Staubli VAL3: isReachable.pgx

program isReachable(pointRx& x_pPoint[], tool x_tTool, bool& x_bUnreached)
  local joint l_jJoint
  local point l_pPoint
begin
  // check the point...
  if pointToJoint(x_tTool,herej(),x_pPoint,l_jJoint)
    x_bUnreached=false
    if size(x_pPoint)>1 and pointToJoint(x_tTool,herej(),x_pPoint[1],l_jJoint)
      x_bUnreached=false
    elseIf size(x_pPoint)>1
      x_bUnreached=true
    endIf
  else
    x_bUnreached=true
  endIf

end
